PROGRAM Motor_Control
VAR
	Process_0: Process;
	Pos: INT;
END_VAR

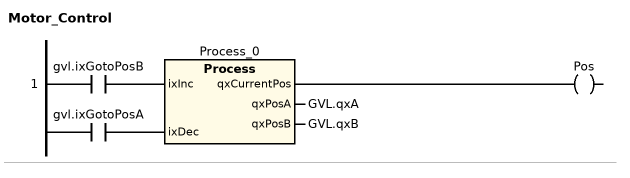
// NETWORK 1
Process_0(ixInc := gvl.ixGotoPosB, ixDec := gvl.ixGotoPosA, qxPosA => GVL.qxA, qxPosB => GVL.qxB); // Process
Pos := Process_0.qxCurrentPos;

END_PROGRAM

(* stored: Version 1.1.0.1, ProductVersion 3.1.4024.12
   POU Motor_Control: Id {97d7822b-b218-4b0c-ac6d-5ebe97b89be2}, SpecialFunc None *)
